PROGRAM MAIN
VAR
	xInput : BOOL;
	xOutput : BOOL;
	
	timer1 : TON;
	timer2 : TON;
END_VAR

xOutput := xInput;

timer1(IN:= NOT timer2.Q, PT:= T#1S);
timer2(IN:= timer1.Q,PT := T#1S);

END_PROGRAM

(* stored: Version 1.1.0.1, ProductVersion 3.1.4024.12
   POU MAIN: Id {c26bae5a-ff24-44e0-b6b0-bc4ad5ea9080}, SpecialFunc None *)
